// TIA Portal project "Blower_Speed_Control" (V19)
// Blower control through speed presets on variable frequency drive

(* hardware
DEVICE "S7-1200 station_1"  S7-1200 Station
   slot 0: "Rack_0"  S7-1200 Rack  Rack  V1.0
   slot 1: "PLC_1"  CPU 1212C AC/DC/Rly  6ES7 212-1BE40-0XB0  V4.6
*)

// ===== PLC "PLC_1"  CPU 1212C AC/DC/Rly =====

VAR_GLOBAL   // PLC tag table "In"
   "Pb_Start" AT %M0.0 : Bool;   // Pushbutton start NO
   "Pb_Stop" AT %M0.1 : Bool;   // Pushbutton stop NC
   "Emergency_Stop" AT %M0.2 : Bool;   // Emergency stop NC
   "Drive_Tripped" AT %M0.3 : Bool;   // Drive tripped contact NO, Logic 1 when drive is in a fault condition
   "Pb_Inc" AT %M0.4 : Bool;   // Pushbutton increment speed
   "Pb_Dec" AT %M0.5 : Bool;   // Pushbutton decrement speed
END_VAR

VAR_GLOBAL   // PLC tag table "Out"
   "Preset_Speed_1" AT %Q0.0 : Bool;   // Preset output one
   "Preset_Speed_2" AT %Q0.1 : Bool;   // Preset output two
   "Preset_Speed_3" AT %Q0.2 : Bool;   // Preset output three
   "Preset_Speed_4" AT %Q0.3 : Bool;   // Preset output four
END_VAR

DATA_BLOCK "Vars"   // DB1
{ S7_Optimized_Access := 'TRUE' }
AUTHOR : Stiven Perez Mora
VERSION : 0.1
   VAR
      Flanco_Start : Bool;
      Flanco_Stop : Bool;
      M_SR : Bool;
      Q_IncDec : Int;
      Flanco_Inc : Bool;
      Flanco_Dec : Bool;
   END_VAR
BEGIN
END_DATA_BLOCK

// folder: System blocks/Program resources

DATA_BLOCK "Timer_Speed_One"   // DB2
{ S7_Optimized_Access := 'TRUE' }
AUTHOR : Simatic
FAMILY : IEC
NAME : IEC_TMR
VERSION : 1.0
// stored: InstanceOfName IEC_TIMER
"IEC_TIMER"
BEGIN
END_DATA_BLOCK

DATA_BLOCK "Timer_Speed_Two"   // DB3
{ S7_Optimized_Access := 'TRUE' }
AUTHOR : Simatic
FAMILY : IEC
NAME : IEC_TMR
VERSION : 1.0
// stored: InstanceOfName IEC_TIMER
"IEC_TIMER"
BEGIN
END_DATA_BLOCK

DATA_BLOCK "Timer_Speed_Three"   // DB4
{ S7_Optimized_Access := 'TRUE' }
AUTHOR : Simatic
FAMILY : IEC
NAME : IEC_TMR
VERSION : 1.0
// stored: InstanceOfName IEC_TIMER
"IEC_TIMER"
BEGIN
END_DATA_BLOCK

DATA_BLOCK "Timer_Speed_Four"   // DB5
{ S7_Optimized_Access := 'TRUE' }
AUTHOR : Simatic
FAMILY : IEC
NAME : IEC_TMR
VERSION : 1.0
// stored: InstanceOfName IEC_TIMER
"IEC_TIMER"
BEGIN
END_DATA_BLOCK

// folder: (top level)

FUNCTION "Increase and Decrease Speed" : Void   // FC1, LAD
TITLE = Increase and Decrease Speed
{ S7_Optimized_Access := 'TRUE' }
AUTHOR : Stiven Perez Mora
VERSION : 0.1
   VAR_INPUT
      Pb_Inc : Bool;
      Pb_Dec : Bool;
   END_VAR
   VAR_OUTPUT
      Speed_One : Bool;
      Speed_Two : Bool;
      Speed_Three : Bool;
   END_VAR
   VAR_IN_OUT
      Speed_Four : Bool;
   END_VAR
   VAR_TEMP   // added for the SCL form of the ladder/FBD networks
      _w1 : Bool;
      _w2 : Bool;
   END_VAR
BEGIN

REGION Network 1: Increase and Decrease Speed
   // Conditions to increase or decrease speed
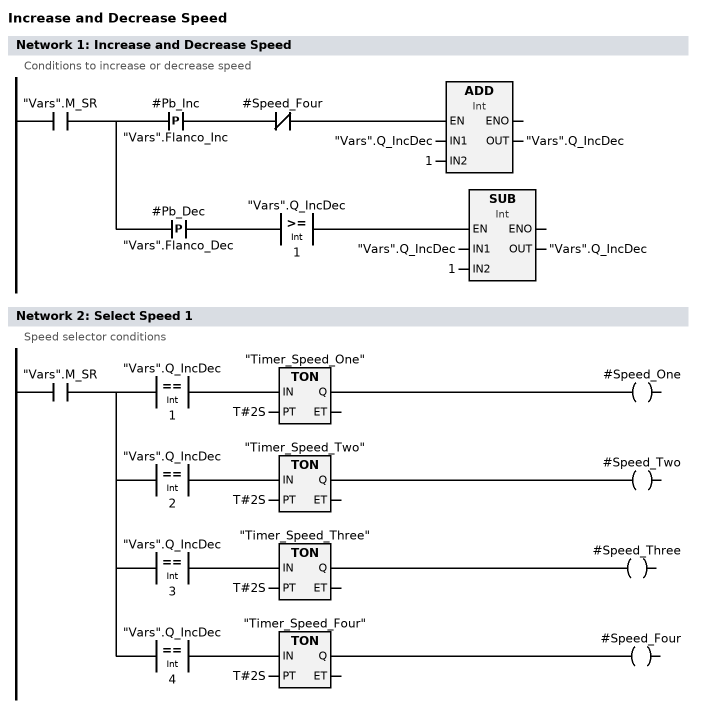
   RUNG wire#powerrail
      Contact( "Vars".M_SR )
      wire#w1
      P_Contact(operand := #Pb_Inc, bit := "Vars".Flanco_Inc)
      I_Contact( #Speed_Four )
      { S7_Templates := "SrcType := Int" } Add(in1 := "Vars".Q_IncDec, in2 := 1, out => "Vars".Q_IncDec)
   END_RUNG
   RUNG wire#w1
      P_Contact(operand := #Pb_Dec, bit := "Vars".Flanco_Dec)
      { S7_Templates := "SrcType := Int" } GE_Contact(in1 := "Vars".Q_IncDec, in2 := 1)
      { S7_Templates := "SrcType := Int" } Sub(in1 := "Vars".Q_IncDec, in2 := 1, out => "Vars".Q_IncDec)
   END_RUNG
   // the same network as SCL:
   #_w1 := "Vars".M_SR AND #Pb_Inc AND NOT "Vars".Flanco_Inc;   // rising edge of #Pb_Inc
   "Vars".Flanco_Inc := #Pb_Inc;
   IF #_w1 AND NOT #Speed_Four THEN "Vars".Q_IncDec := "Vars".Q_IncDec + 1; END_IF;
   #_w2 := "Vars".M_SR AND #Pb_Dec AND NOT "Vars".Flanco_Dec;   // rising edge of #Pb_Dec
   "Vars".Flanco_Dec := #Pb_Dec;
   IF #_w2 AND ("Vars".Q_IncDec >= 1) THEN "Vars".Q_IncDec := "Vars".Q_IncDec - 1; END_IF;
END_REGION

REGION Network 2: Select Speed 1
   // Speed selector conditions
   "Timer_Speed_One".TON(IN := "Vars".M_SR AND ("Vars".Q_IncDec = 1), PT := T#2S);
   #Speed_One := "Timer_Speed_One".Q;
   "Timer_Speed_Two".TON(IN := "Vars".M_SR AND ("Vars".Q_IncDec = 2), PT := T#2S);
   #Speed_Two := "Timer_Speed_Two".Q;
   "Timer_Speed_Three".TON(IN := "Vars".M_SR AND ("Vars".Q_IncDec = 3), PT := T#2S);
   #Speed_Three := "Timer_Speed_Three".Q;
   "Timer_Speed_Four".TON(IN := "Vars".M_SR AND ("Vars".Q_IncDec = 4), PT := T#2S);
   #Speed_Four := "Timer_Speed_Four".Q;
END_REGION
END_FUNCTION

FUNCTION "Start Stop Process" : Void   // FC2, LAD
{ S7_Optimized_Access := 'TRUE' }
AUTHOR : Stiven Perez Mora
VERSION : 0.1
   VAR_INPUT
      Pb_Start : Bool;
      Pb_Stop : Bool;
      Emergency_Stop : Bool;
   END_VAR
   VAR_TEMP   // added for the SCL form of the ladder/FBD networks
      _w1 : Bool;
   END_VAR
BEGIN

REGION Network 1: Start Process
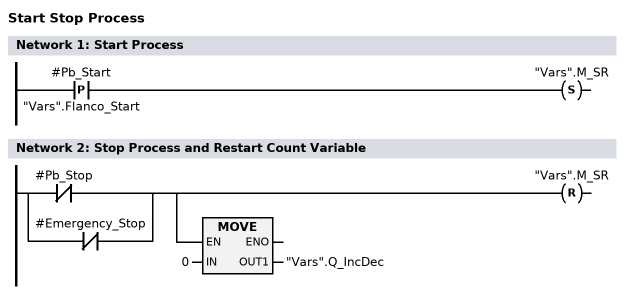
   RUNG wire#powerrail
      P_Contact(operand := #Pb_Start, bit := "Vars".Flanco_Start)
      S_Coil( "Vars".M_SR )
   END_RUNG
   // the same network as SCL:
   #_w1 := #Pb_Start AND NOT "Vars".Flanco_Start;   // rising edge of #Pb_Start
   "Vars".Flanco_Start := #Pb_Start;
   IF #_w1 THEN "Vars".M_SR := TRUE; END_IF;
END_REGION

REGION Network 2: Stop Process and Restart Count Variable
   RUNG wire#powerrail
      I_Contact( #Pb_Stop )
      wire#w1
      R_Coil( "Vars".M_SR )
   END_RUNG
   RUNG wire#powerrail
      I_Contact( #Emergency_Stop )
   END_RUNG wire#w1
   RUNG wire#w1
      Move(in := 0, out1 => "Vars".Q_IncDec)
   END_RUNG
   // the same network as SCL:
   IF NOT #Pb_Stop OR NOT #Emergency_Stop THEN
       "Vars".M_SR := FALSE;
       "Vars".Q_IncDec := 0;
   END_IF;
END_REGION
END_FUNCTION

ORGANIZATION_BLOCK "Main"   // OB1, LAD, ProgramCycle
TITLE = "Main Program Sweep (Cycle)"
{ S7_Optimized_Access := 'TRUE' }
VERSION : 0.1
   VAR_INPUT
      Initial_Call : Bool;   // Initial call of this OB
      Remanence : Bool;   // =True, if remanent data are available
   END_VAR
BEGIN

REGION Network 1: Start Stop Process Block
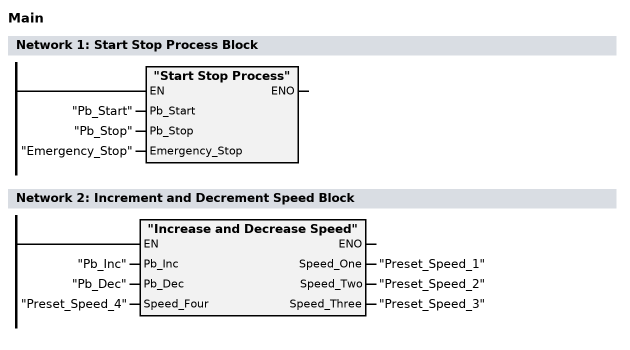
   RUNG wire#powerrail
      "Start Stop Process"(Pb_Start := "Pb_Start", Pb_Stop := "Pb_Stop", Emergency_Stop := "Emergency_Stop")
   END_RUNG
   // the same network as SCL:
   "Start Stop Process"(Pb_Start := "Pb_Start", Pb_Stop := "Pb_Stop", Emergency_Stop := "Emergency_Stop");
END_REGION

REGION Network 2: Increment and Decrement Speed Block
   RUNG wire#powerrail
      "Increase and Decrease Speed"(Pb_Inc := "Pb_Inc", Pb_Dec := "Pb_Dec", Speed_One => "Preset_Speed_1", Speed_Four := "Preset_Speed_4", Speed_Two => "Preset_Speed_2", Speed_Three => "Preset_Speed_3")
   END_RUNG
   // the same network as SCL:
   "Increase and Decrease Speed"(Pb_Inc := "Pb_Inc",
                           Pb_Dec := "Pb_Dec",
                           Speed_Four := "Preset_Speed_4",
                           Speed_One => "Preset_Speed_1",
                           Speed_Two => "Preset_Speed_2",
                           Speed_Three => "Preset_Speed_3");
END_REGION
END_ORGANIZATION_BLOCK